FUNCTION_BLOCK MotorProtection
VAR_INPUT
END_VAR
VAR_OUTPUT
END_VAR
VAR
	xInputAddress AT %I* : BIT;
	bOvercurrentStatus : BOOL;
END_VAR

METHOD FB_init : BOOL
VAR_INPUT
	bInitRetains : BOOL; // if TRUE, the retain variables are initialized (warm start / cold start)
	bInCopyCode : BOOL;  // if TRUE, the instance afterwards gets moved into the copy code (online change)
END_VAR
END_METHOD

PROPERTY PUBLIC overcurrentStatus : BOOL
GET
overcurrentStatus := bOvercurrentStatus;
END_GET
END_PROPERTY

END_FUNCTION_BLOCK

(* stored: Version 1.1.0.1, ProductVersion 3.1.4024.12
   POU MotorProtection: Id {e46a7c32-9a2e-4c40-a832-d9bb44fbf82d}, SpecialFunc None
   Method FB_init: Id {ceb897a8-8b62-4dfb-9e7e-686da1b4332b}
   Property overcurrentStatus: Id {fd63a1f7-1f8a-46e0-9418-04316c5a36c2}
   Get Get: Id {d8aa0b07-2a7d-45c2-86b7-2fb56ee8f90e} *)
